// TIA Portal V19 export
VAR_GLOBAL   // PLC tag table "LB113"
   LB113_JB_Cut_Lp_Cycle AT %Q116.5 : Bool;   // 326SH2
   LB113_JB_Cut_Pb_Cycle AT %I119.1 : Bool;   // 326SH2
   LB113_JB_EntryClamp_Sel_Close AT %I120.6 : Bool;   // 327SA2
   LB113_JB_EntryClamp_Sel_Open AT %I120.5 : Bool;   // 327SA1
   LB113_JB_ExitClamp_Sel_Close AT %I119.7 : Bool;   // 326SA2
   LB113_JB_ExitClamp_Sel_Open AT %I119.6 : Bool;   // 326SA2
   LB113_JB_Lp_AtRest AT %Q117.5 : Bool;   // 328HL1
   LB113_JB_Pichroll_Pb_Bwd AT %I119.5 : Bool;   // 326SH4
   LB113_JB_Pichroll_Pb_Fwd AT %I119.4 : Bool;   // 326SH3
   LB113_JB_Pinchroll_Lp_Bwd AT %Q116.7 : Bool;   // 326SH4
   LB113_JB_Pinchroll_Lp_Fwd AT %Q116.6 : Bool;   // 326SH3
   LB113_JB_Torch_Lp_Bwd AT %Q117.4 : Bool;   // 327SH5
   LB113_JB_Torch_Lp_Fwd AT %Q117.3 : Bool;   // 327SH4
   LB113_JB_Torch_Pb_Bwd AT %I120.4 : Bool;   // 327SH5
   LB113_JB_Torch_Pb_Fwd AT %I120.3 : Bool;   // 327SH4
   LB113_JB_Weld_Lp_Cycle AT %Q117.0 : Bool;   // 327SH2
   LB113_JB_Weld_Lp_Man AT %Q117.1 : Bool;   // 327SH1
   LB113_JB_Weld_Pb_Cycle AT %I120.0 : Bool;   // 327SH1
   LB113_JB_Weld_Pb_Man AT %I120.1 : Bool;   // 327SH2
   LB113_Lp_ExtraLow AT %Q117.2 : Bool;   // 327SH3
   LB113_Lp_Provino AT %Q116.4 : Bool;   // 326SH1
   LB113_Pb_ExtraLow AT %I120.2 : Bool;   // 327SH3
   LB113_Pb_Provino AT %I119.0 : Bool;   // 326SH1
   LB113_PinchRoll_Sel_Close AT %I119.3 : Bool;   // 326SA2
   LB113_PinchRoll_Sel_Open AT %I119.2 : Bool;   // 326SA1
   LB113_Straightener_Lp_Bwd AT %Q117.7 : Bool;   // 328HL3
   LB113_Straightener_Lp_Fwd AT %Q117.6 : Bool;   // 328HL2
   LB113_Straightener_Pb_Bwd AT %I121.0 : Bool;   // 328SH2
   LB113_Straightener_Pb_Fwd AT %I120.7 : Bool;   // 328SH1
   LB113_Button_L AT %I1034.2 : Bool;   // 104DI2 - 201SB1
   LB113_DeadMan_Ch1 AT %I1034.3 : Bool;   // 104DI3 - 201SB3
   LB113_DeadMan_Ch2 AT %I1034.7 : Bool;   // 104DI7 - 201SB3
   LB113_Button_R AT %I1034.6 : Bool;   // 104DI6 - 201SB2
END_VAR
